FUNCTION_BLOCK FB_PlanarXtsMover

VAR_INPUT
	iTcIoXtsXpuMover			: REFERENCE TO Tc3_XTS_Utility.I_TcIoXtsXpuMover;
END_VAR

VAR
	stMoverOptions						: ST_MoverOptions;
	BaseMoveOptions						: Tc3_Mc3PlanarMotion.ST_MoveOnTrackOptions;
	GearInMasterMoverOptions	: Tc3_Mc3PlanarMotion.ST_GearInPosOnTrackWithMasterMoverOptions;
	
	MC_PlanarFeedbackGearInPosOnTrackWithMasterMover : Tc3_Mc3PlanarMotion.MC_PlanarFeedbackGearInPosOnTrackWithMasterMover;
		
	nMoverId			    				: UDINT;
	
	MoverFeedback							: Tc3_Mc3PlanarMotion.MC_PlanarFeedback;

	_McPlanarMover						: Tc3_Mc3PlanarMotion.MC_PlanarMover;
	_McPlanarTrackTrail    		: Tc3_Mc3PlanarMotion.MC_PlanarTrackTrail;
                        		
	stXtsPositionInfo					: Tc3_XTS_Utility.ST_PositionInfo;
	                      		
	Physics										: Tc3_Physics.PositionXYC;
	Dynamics									: Tc3_Physics.DynamicConstraint_PathXY;

	Mover				        			: MoverSort;
	
	SyncTrail 								: Tc3_Mc3PlanarMotion.MC_PlanarTrackTrail; 
	
	CmdDivert									: BOOL;
	eMerge										: E_MergeType;
	//InSync										: BOOL;
END_VAR

METHOD FB_init : BOOL
VAR_INPUT
	bInitRetains : BOOL; // if TRUE, the retain variables are initialized (warm start / cold start)
	bInCopyCode : BOOL;  // if TRUE, the instance afterwards gets moved into the copy code (online change)
END_VAR
stMoverOptions.BaseMoveOptions REF= BaseMoveOptions;
stMoverOptions.GearInMasterMoverOptions	REF= GearInMasterMoverOptions;

//Most options already initialized
//GearInMasterMoverOptions.allowedSlaveSyncDirections 				:= MC_SYNC_DIRECTIONS.Positive;
//GearInMasterMoverOptions.directionMasterSyncPosition				:= Tc3_Mc3PlanarMotion.MC_DIRECTION.mcDirectionNonModulo;
//GearInMasterMoverOptions.directionSlaveSyncPosition					:= Tc3_Mc3PlanarMotion.MC_DIRECTION.mcDirectionNonModulo;
//GearInMasterMoverOptions.followMover												:= FALSE;
GearInMasterMoverOptions.gap 																:= BaseMoveOptions.gap;
//GearInMasterMoverOptions.inSyncToleranceDistance						:= 0;
//GearInMasterMoverOptions.moduloToleranceMasterSyncPosition	:= 0;
//GearInMasterMoverOptions.moduloToleranceSlaveSyncPosition		:= 0;

syncTrail.AddTrack(track:= GVL_Mc3.MC_Tracks[E_TrackNum.Small]); 
syncTrail.AddTrack(track:= GVL_Mc3.MC_Tracks[E_TrackNum.Main]);
END_METHOD

METHOD Init : BOOL
VAR_INPUT

	XtsMover:   I_XtsXlMover1;
	XtsProcessingUnit :  I_XtsProcessingUnit1;
END_VAR



ipXtsMover:= XtsMover;
ipXtsProcessingUnit :=  XtsProcessingUnit;

stMoveOnTrackOptions.direction := MC_Direction.mcDirectionPositive;
stMoveOnTrackOptions.gapMode := MC_GAP_MODE_ON_TRACK.Fast1D;
stMoveOnTrackOptions.gap:= 800;

syncTrail.AddTrack(track:= GVL_Mc.MC_Tracks[E_TrackNum.Small]); 
syncTrail.AddTrack(track:= GVL_Mc.MC_Tracks[E_TrackNum.Main]); 


//_stDynamics.SetValuesVADJ(500, 4000, 4000, 10000);

bIsInitialized := TRUE;
END_METHOD

PROPERTY IsCommandedInShortcut : BOOL
GET
VAR
	nCounter: UDINT := 0;
END_VAR
_mcPlanarMover.GetTrackTrailInformation(_PlanarTrail);

IF _PlanarTrail.Error OR _PlanarTrail.Size < 1 THEN
   IsCommandedInShortcut := FALSE;
   RETURN;
END_IF
   
FOR nCounter := 0 TO _PlanarTrail.Size - 1 DO
	IF _PlanarTrail.GetTrackOidAt(nCounter) = GVL_Mc3.MC_Tracks[E_TrackNum.Small].MCTOPLC_STD.TrackOID  THEN
		IsCommandedInShortcut := TRUE;
		RETURN;
	END_IF
END_FOR

IsCommandedInShortcut := FALSE;
END_GET
END_PROPERTY

METHOD JoinTrack

VAR_INPUT
	feedback: REFERENCE TO MC_PlanarFeedback;
END_VAR

VAR_IN_OUT
	track: MC_PlanarTrack;
END_VAR
_McPlanarMover.JoinTrack(feedback, track, 0, 0);
END_METHOD

METHOD M_EvaluateGap
VAR_INPUT
	MoverIndex	: UDINT;
END_VAR
IF TrackSectors[MoverIndex].SectorStatus[GC.OUTER_TIGHTGAP_ZONE].MoverIsOnSector OR
TrackSectors[MoverIndex].SectorStatus[GC.INNER_MERGE_TO_FINISH].MoverIsOnSector THEN
	fbPlanarXtsMover[MoverIndex].P_MoverOptions.BaseMoveOptions.gap := stMoverConfig.TightMoverGap;
ELSIF TrackSectors[MoverIndex].SectorStatus[GC.OUTER_PRE_TG_ZONE].MoverIsOnSector THEN
	fbPlanarXtsMover[MoverIndex].P_MoverOptions.TempGap := HelperFunctions.F_MapLReal(x := TrackSectors[MoverIndex].SectorStatus[GC.OUTER_PRE_TG_ZONE].PercentOfSectorTraversed,
														in_min := 0.0, in_max := 1.0, out_min := stMoverConfig.NormalMoverGap, out_max := stMoverConfig.TightMoverGap);
	fbPlanarXtsMover[MoverIndex].P_MoverOptions.BaseMoveOptions.gap := fbPlanarXtsMover[MoverIndex].P_MoverOptions.TempGap;
ELSIF TrackSectors[MoverIndex].SectorStatus[GC.OUTER_POST_TG_ZONE].MoverIsOnSector THEN
	fbPlanarXtsMover[MoverIndex].P_MoverOptions.TempGap := HelperFunctions.F_MapLReal(x := TrackSectors[MoverIndex].SectorStatus[GC.OUTER_POST_TG_ZONE].PercentOfSectorTraversed,
														in_min := 0.0, in_max := 1.0, out_min := stMoverConfig.TightMoverGap, out_max := stMoverConfig.NormalMoverGap);
	fbPlanarXtsMover[MoverIndex].P_MoverOptions.BaseMoveOptions.gap := fbPlanarXtsMover[MoverIndex].P_MoverOptions.TempGap;
ELSE
	fbPlanarXtsMover[MoverIndex].P_MoverOptions.BaseMoveOptions.gap := stMoverConfig.NormalMoverGap;
END_IF

IF fbPlanarXtsMover[MoverIndex].P_MoverOptions.BaseMoveOptions.gap = stMoverConfig.NormalMoverGap OR
	fbPlanarXtsMover[MoverIndex].P_MoverOptions.BaseMoveOptions.gap = stMoverConfig.TightMoverGap THEN
	fbPlanarXtsMover[MoverIndex].P_MoverOptions.GapInTransition := FALSE;
ELSE
	fbPlanarXtsMover[MoverIndex].P_MoverOptions.GapInTransition := TRUE;
END_IF
END_METHOD

PROPERTY P_CmdDivert : REFERENCE TO BOOL
GET
P_CmdDivert	REF= CmdDivert;
END_GET
END_PROPERTY

PROPERTY P_Dynamics : REFERENCE TO Tc3_Physics.DynamicConstraint_PathXY
GET
P_Dynamics	REF= Dynamics;
END_GET
END_PROPERTY

PROPERTY P_eMerge : REFERENCE TO E_MergeType
GET
P_eMerge	REF= eMerge;
END_GET
END_PROPERTY

PROPERTY P_InSync : REFERENCE TO BOOL
GET
P_InSync REF= MC_PlanarFeedbackGearInPosOnTrackWithMasterMover.inSync;
END_GET
END_PROPERTY

PROPERTY P_MC_PlanarMover : REFERENCE TO Tc3_Mc3PlanarMotion.MC_PlanarMover
GET
P_MC_PlanarMover REF= _McPlanarMover;
END_GET
END_PROPERTY

PROPERTY P_MoverFeedback : REFERENCE TO Tc3_Mc3PlanarMotion.MC_PlanarFeedback
GET
P_MoverFeedback REF= MoverFeedback;
END_GET
END_PROPERTY

PROPERTY P_MoverId : UDINT
GET
P_MoverId	:= nMoverId;
END_GET
SET
nMoverId := P_MoverId;
END_SET
END_PROPERTY

PROPERTY P_MoverOptions : REFERENCE TO ST_MoverOptions
GET
P_MoverOptions REF= stMoverOptions;
END_GET
END_PROPERTY

PROPERTY P_MoverSort : REFERENCE TO MoverSort
GET
P_MoverSort	REF= Mover;
END_GET
END_PROPERTY

PROPERTY P_Physics : REFERENCE TO Tc3_Physics.PositionXYC
GET
P_Physics	REF= Physics;
END_GET
END_PROPERTY

PROPERTY P_PlanarFeedbackGearMM : REFERENCE TO Tc3_Mc3PlanarMotion.MC_PlanarFeedbackGearInPosOnTrackWithMasterMover
GET
P_PlanarFeedbackGearMM REF= MC_PlanarFeedbackGearInPosOnTrackWithMasterMover;
END_GET
END_PROPERTY

PROPERTY P_SyncTrail : REFERENCE TO Tc3_Mc3PlanarMotion.MC_PlanarTrackTrail
GET
P_SyncTrail REF= SyncTrail;
END_GET
END_PROPERTY

PROPERTY P_TrackConfig : REFERENCE TO ST_TrackConfig
GET
END_GET
END_PROPERTY

PROPERTY P_XtsPositionInfo : REFERENCE TO Tc3_XTS_Utility.ST_PositionInfo
GET
P_XtsPositionInfo	REF= stXtsPositionInfo;
END_GET
END_PROPERTY

METHOD SyncToOtherMover : BOOL
VAR_INPUT
	masterSyncPos : LREAL; // Position on the master track
	followerSyncPos : LREAL; // position on the follower track
	PlanarMoverToFollow: REFERENCE TO Tc3_Mc3PlanarMotion.MC_PlanarMover;
	masterTrack : REFERENCE TO Tc3_Mc3PlanarMotion.MC_PlanarTrack; 
	followerTrack : REFERENCE TO Tc3_Mc3PlanarMotion.MC_PlanarTrack; 
	velo : LREAL; 
END_VAR

VAR
	trail: Tc3_Mc3PlanarMotion.MC_PlanarTrackTrail;

END_VAR
//Options.allowedSlaveSyncDirections := MC_SYNC_DIRECTIONS.Positive; 
//options.directionMasterSyncPosition := MC_DIRECTION.mcDirectionNonModulo; 
//options.directionSlaveSyncPosition := MC_DIRECTION.mcDirectionNonModulo;  
//options.followMover := FALSE; 
//options.gap := 0; // elimnate gap funciton 
//options.inSyncToleranceDistance :=0; 
//options.moduloToleranceMasterSyncPosition := 0; 
//options.moduloToleranceSlaveSyncPosition := 0;  
//_stDynamics.V := velo; 

fbPlanarMover.GearInPosOnTrackWithMasterMover(
//	commandFeedback:=  SyncMoverFeedback , 
//	masterMover:= PlanarMoverToFollow , 
//	trackTrail:= syncTrail, // may need to give a trail maybe not
//	masterSyncPosition:= masterSyncPos, 
//	masterSyncPositionTrack:= MasterTrack , 
//	slaveSyncPosition:= followerSyncPos, 
//	slaveSyncPositionTrack:= followerTrack, 
//	constraint:=_stDynamics , 
//	options:=options );
END_METHOD

METHOD Update : PVOID
IF iTcIoXtsXpuMover <> 0 THEN
  stXtsPositionInfo	:= iTcIoXtsXpuMover.GetPositionInfo();
END_IF

_mcPlanarMover.Update();

IF eMerge <> E_MergeType.NoMerge THEN
	MC_PlanarFeedbackGearInPosOnTrackWithMasterMover.Update();
END_IF

_mcPlanarMover.GetTrackTrailInformation(_McPlanarTrackTrail);

Mover.MoverNumber 	:= nMoverId;
Mover.MoverPos    	:= _McPlanarMover.MCTOPLC.SETONTRACK.SetPos;
Mover.TrackID     	:= _McPlanarMover.MCTOPLC.SETONTRACK.TrackOID;
//MoverPhysics		:= 

{warning <'Method Not Called'>}
//_M_UpdateStatus();

IF _McPlanarTrackTrail.Error OR _McPlanarTrackTrail.Size <= 1 THEN
   RETURN;
END_IF

IF iTcIoXtsXpuMover <> 0 THEN
  //SmallCircle
  IF _McPlanarTrackTrail.GetTrackOidAt(1) = MC_Tracks[E_TrackNum.Small].MCTOPLC_STD.TrackOID   THEN
    iTcIoXtsXpuMover.SetActiveTrackObjectId(XtsCompleteTrackInnerOID);
  //BigCircle
  ELSIF _McPlanarTrackTrail.GetTrackOidAt(1) =MC_Tracks[E_TrackNum.Big].MCTOPLC_STD.TrackOID THEN
    iTcIoXtsXpuMover.SetActiveTrackObjectId(XtsCompleteTrackOuterOID);
  END_IF
END_IF
END_METHOD

END_FUNCTION_BLOCK

(* stored: Version 1.1.0.1
   POU FB_PlanarXtsMover: Id {e98e5f10-cdde-43fc-96da-1ae5f511366a}, SpecialFunc None
   Folder Methods: Id {497e6300-3e6d-49b8-a318-13b94b960f56}
   Folder Properties: Id {bafe569f-b5f0-4de9-ae48-854cd11ccd2e}
   Method FB_init: Id {4b084dbd-ec42-0e10-3862-f9a7de67a652}
   Method Init: Id {6ea09207-c20a-09f4-120c-5892eef487d3}
   Property IsCommandedInShortcut: Id {e5e69e7e-f163-4728-82da-b10e582ce622}
   Get Get: Id {7a71ba46-249d-415a-b1f4-f1c52c07bed0}
   Method JoinTrack: Id {fd819ce6-c064-4bae-aa84-926325f13c12}
   Method M_EvaluateGap: Id {fcb9e531-850f-006f-2c28-ec403292155f}
   Property P_CmdDivert: Id {8cede827-2b25-094d-2c84-715767aaf20f}
   Get Get: Id {ee22a2e2-25c9-085f-3a80-3e499cb6195c}
   Property P_Dynamics: Id {012820e2-39fa-01ed-0dfe-860675d63f58}
   Get Get: Id {985c286c-7fa7-0076-0f00-c12e68aed781}
   Property P_eMerge: Id {5698d2c6-a9ba-0594-1fa9-f7ecaefdee80}
   Get Get: Id {b80825a0-b14e-0969-14a3-bf841bda528e}
   Property P_InSync: Id {2df9b0c6-84c0-0064-0364-e2a3e9418875}
   Get Get: Id {d847e18f-6401-0e3b-14bd-4b43c4d4c8c5}
   Property P_MC_PlanarMover: Id {79d72b75-52b9-47c8-886e-5e60276bf5f1}
   Get Get: Id {71cad725-c4c4-49c5-9410-cee17b681f5a}
   Property P_MoverFeedback: Id {02ef7bc1-889e-07f7-3c27-62976c319346}
   Get Get: Id {159a251f-157e-010b-1c51-0b1d7364f59a}
   Property P_MoverId: Id {033bc7d6-a908-0af3-1630-2fc499f56ad8}
   Get Get: Id {c0e5d564-a073-06e0-3bca-52836c21275c}
   Set Set: Id {ff03ecba-f79d-0c21-3b65-7c6a4248584c}
   Property P_MoverOptions: Id {fb098007-5ff7-07f5-0b7d-758e50c8b22a}
   Get Get: Id {9944f816-4bb0-07d5-02b6-9a4f523da06d}
   Property P_MoverSort: Id {a5ac8d37-9108-0740-305c-d3b342270158}
   Get Get: Id {bae1975d-f945-0652-3748-976b73c4f7d6}
   Property P_Physics: Id {056b1259-392a-0821-097b-b08bee10a569}
   Get Get: Id {e7ba31e5-6730-0d69-35c1-51b7d57fd5fd}
   Property P_PlanarFeedbackGearMM: Id {d729f8fd-3179-0343-3353-ddd710f91bdd}
   Get Get: Id {2b88ac50-2312-0cef-1014-00a094a686f4}
   Property P_SyncTrail: Id {317f6011-5dc7-037e-1a7f-22f5a06871b8}
   Get Get: Id {19b14c75-2123-015f-13bf-ec8c0b82eace}
   Property P_TrackConfig: Id {e32b61fd-1607-0d8a-3b00-a92d697c1e42}
   Get Get: Id {f2020383-ba74-08e6-01f4-c80f3d2580af}
   Property P_XtsPositionInfo: Id {eee46ce5-009e-038a-12e5-cdbf8f2886af}
   Get Get: Id {58ff9574-093b-05dd-3592-27328f83735e}
   Method SyncToOtherMover: Id {f3ce074a-da58-0d33-2eed-617bf65f1455}
   Method Update: Id {2a189ea7-97f2-4dc0-980a-fdde9c091766} *)
